{attribute 'qualified_only'}
VAR_GLOBAL CONSTANT
	STR_SIZE : FsT_Size := 80; // Size of general string.
	SSTR_SIZE : FsT_Size := 40; // Size of short string.
	LSTR_SIZE : FsT_Size := 255; // Size of long string.
	INFO_SCAN_SIZE : FsT_Size := 15000; // How many bytes to scan when looking for information. e.g. it's FsFB_Object to find the size of a child object in static memory.
END_VAR

(* stored: Version 1.1.0.1, ProductVersion 3.1.4024.4
   GVL FsParam_Core: Id {23f779d3-74b3-4231-a330-7fe9e566b126}, ParameterList True *)
